//The return value is not evaluated. For a specific influence, you can also declare the

//methods explicitly and provide additional code there with the standard initialization

//code. You can evaluate the return value.
METHOD FB_Init : BOOL
VAR_INPUT
	bInitRetains : BOOL; // TRUE: the retain variables are initialized (reset warm / reset cold)
	bInCopyCode	 : BOOL; // TRUE: the instance will be copied to the copy code afterward (online change)  
	Dimensions	 : I_SingleDimensionZone;
END_VAR
_Dimensions := Dimensions;
END_METHOD

METHOD IsMoverInPosition : BOOL
VAR_INPUT
	Mover : I_XtsMover;
END_VAR

VAR
	startPosition : LREAL;
	endPosition	  : LREAL;
	tmp : LREAL;
END_VAR
startPosition := _Dimensions.StartPosition;
endPosition	  := _Dimensions.EndPosition;
IF Mover.Status.CurrentTrack.Length <> 0 THEN
	startPosition := startPosition - Mover.Status.CurrentTrack.Length * TRUNC(_Dimensions.StartPosition / Mover.Status.CurrentTrack.Length);
	IF startPosition < 0.0 THEN
		startPosition := startPosition + Mover.Status.CurrentTrack.Length;
	END_IF

	endPosition := endPosition - Mover.Status.CurrentTrack.Length * TRUNC(_Dimensions.EndPosition / Mover.Status.CurrentTrack.Length);
	IF endPosition < 0.0 THEN
		endPosition := endPosition + Mover.Status.CurrentTrack.Length;
	END_IF
END_IF

IF startPosition < endPosition THEN
	IsMoverInPosition := Mover.Position > startPosition AND Mover.Position < endPosition;
ELSE
	IsMoverInPosition := Mover.Position > startPosition OR Mover.Position < endPosition;
END_IF
END_METHOD

END_FUNCTION_BLOCK

// _Internal/Zone/Interfaces/I_MoverInPositionChecker
INTERFACE I_MoverInPositionChecker EXTENDS I_Base

METHOD IsMoverInPosition : BOOL
VAR_INPUT
	Mover : I_XtsMover;
END_VAR
END_METHOD

END_INTERFACE

// _Internal/Zone/MoverZoneDistanceComparer
{attribute 'no_explicit_call' := 'This FB is a CLASS and must be accessed using methods or properties'}
{attribute 'conditional_show'}
FUNCTION_BLOCK MoverZoneDistanceComparer IMPLEMENTS I_XtsMoverComparer
VAR
	_ZoneDimensions : I_SingleDimensionZone;
END_VAR

METHOD Compare : SINT
VAR_INPUT
	Mover1 : I_XtsMover;
	Mover2 : I_XtsMover;
END_VAR

VAR
	Mover1Distance : LREAL;
	Mover2Distance : LREAL;
END_VAR
Mover1Distance := MoverDistance(_ZoneDimensions.StartPosition, Mover1.Position, Mover1.Status.CurrentTrack.Length);
Mover2Distance := MoverDistance(_ZoneDimensions.StartPosition, Mover2.Position, Mover2.Status.CurrentTrack.Length);
IF Mover1Distance < Mover2Distance THEN
	Compare := -1;
ELSIF Mover1Distance > Mover2Distance THEN
	Compare := 1;
ELSE
	Compare := 0;
END_IF
END_METHOD

//FB_Init is always available implicitly and it is used primarily for initialization.
//The return value is not evaluated. For a specific influence, you can also declare the
//methods explicitly and provide additional code there with the standard initialization
//code. You can evaluate the return value.
METHOD FB_Init: BOOL
VAR_INPUT
    bInitRetains: BOOL; // TRUE: the retain variables are initialized (reset warm / reset cold)
    bInCopyCode: BOOL;  // TRUE: the instance will be copied to the copy code afterward (online change)   
	Dimensions : I_SingleDimensionZone;
END_VAR
_ZoneDimensions := Dimensions;
END_METHOD

END_FUNCTION_BLOCK

// _Internal/Zone/Interfaces/I_XtsMoverComparer
INTERFACE I_XtsMoverComparer EXTENDS I_Base

METHOD Compare : SINT
VAR_INPUT
	Mover1 : I_XtsMover;
	Mover2 : I_XtsMover;
END_VAR
END_METHOD

END_INTERFACE

// _Internal/Zone/MoverDistance
FUNCTION MoverDistance : LREAL
VAR_INPUT
	StartPosition : LREAL;
	MoverPosition : LREAL;
	TrackLength	  : LREAL;
END_VAR

VAR
	NormalizedStart : LREAL;
	Distance		: LREAL;
END_VAR

IF TrackLength = 0 THEN
	MoverDistance := 0;
	RETURN;
END_IF

NormalizedStart := StartPosition - TrackLength * TRUNC(StartPosition / TrackLength);
IF normalizedStart < 0 THEN
	NormalizedStart := NormalizedStart + TrackLength;
END_IF;

Distance := MoverPosition - NormalizedStart;
IF Distance < 0 THEN
	Distance := Distance + TrackLength;
END_IF;

MoverDistance := Distance;

END_FUNCTION

// _Internal/Zone/ZoneMonitor
{attribute 'no_explicit_call' := 'This FB is a CLASS and must be accessed using methods or properties'}
{attribute 'conditional_show'}
FUNCTION_BLOCK ZoneMonitor IMPLEMENTS I_ZoneMonitor
VAR
	_DefaultCurrentMovers : XtsMoverList;
	_CurrentMovers		  : I_XtsMoverList := _DefaultCurrentMovers;
	_MoverChecker		  : I_MoverInPositionChecker;
	_MonitoredMovers	  : I_XtsMoverCollection;
	_ZoneComparer		  : I_XtsMoverComparer;
	_ZoneDimensions		  : I_SingleDimensionZone;
	_Logger				  : I_MechatronicsLogger;
	LogSource			  : TraceSourceInfo;
	LogMessage			  : TraceMessageInfo;
END_VAR

METHOD CyclicLogic
VAR
	Mover				   : I_XtsMover;
	inPosition			   : BOOL;
	inCollection		   : BOOL;
	additionIndex		   : UDINT;
	CompareResults		   : SINT;
	EntranceEvent		   : E_ThresholdEvent;
	ExitEvent			   : E_ThresholdEvent;
	ThresholdEventOccurred : BOOL;
END_VAR
_MonitoredMovers.ResetIterator();
WHILE _MonitoredMovers.MoveToNext DO
	__QUERYINTERFACE(_MonitoredMovers.Current, Mover);
	IF Mover.Status.CurrentTrack.Length = 0 THEN
		LogMessage.MessageId := E_XtsLogMessage.ZoneMoverErrorTrackLengthZero;
		LogMessage.Severity	 := 3;
		_Logger.LogMessageInstance(LogSource, LogMessage);
		CONTINUE;
	END_IF

	inPosition := _MoverChecker.IsMoverInPosition(Mover);

	//Need to check if crossed the threshold of the exit or the entrance
	EntranceEvent		   := CheckForThresholdEvent(Mover, _ZoneDimensions.StartPosition);
	ExitEvent			   := CheckForThresholdEvent(Mover, _ZoneDimensions.EndPosition);
	ThresholdEventOccurred := (EntranceEvent <> E_ThresholdEvent.NoEvent) AND (ExitEvent <> E_ThresholdEvent.NoEvent);
	inCollection		   := _CurrentMovers.Contains(Mover);
	IF NOT inPosition AND inCollection THEN
		_CurrentMovers.Remove(Mover);
		CONTINUE;
	END_IF

	//Adds the Mover into the collection sorted by Position Descending
	IF inPosition AND NOT inCollection THEN
		_CurrentMovers.ResetIterator();
		WHILE _CurrentMovers.MoveToNext DO
			CompareResults := _ZoneComparer.Compare(Mover, _CurrentMovers.Current);
			IF CompareResults < 0 THEN //Mover 1 is closer to Start
				additionIndex := _CurrentMovers.CurrentItem - 1;
				EXIT;
			ELSIF CompareResults > 0 THEN //Mover 2 is closer to Start
				additionIndex := _CurrentMovers.CurrentItem;
			ELSE //Movers are equadistant, should never happen. Only realistically happens if TrackLength = 0

				//
			END_IF
		END_WHILE

		_CurrentMovers.InsertAtIndex(Mover, additionIndex);
	ELSIF ThresholdEventOccurred AND inCollection THEN
		(*Search the Collection to find the new index
			Remove from old index
			Add to new*)
		_CurrentMovers.ResetIterator();
		WHILE _CurrentMovers.MoveToNext DO
			CompareResults := _ZoneComparer.Compare(Mover, _CurrentMovers.Current);
			IF CompareResults < 0 THEN //Mover 1 is closer to Start
				additionIndex := _CurrentMovers.CurrentItem - 1;
				EXIT;
			ELSIF CompareResults > 0 THEN //Mover 2 is closer to Start
				additionIndex := _CurrentMovers.CurrentItem;
			ELSE //Movers are equadistant, should never happen. Only realistically happens if TrackLength = 0

				//
			END_IF
		END_WHILE

		_CurrentMovers.Remove(Mover);
		_CurrentMovers.InsertAtIndex(Mover, additionIndex);
	END_IF
END_WHILE
END_METHOD

//FB_Init is always available implicitly and it is used primarily for initialization.

//The return value is not evaluated. For a specific influence, you can also declare the

//methods explicitly and provide additional code there with the standard initialization

//code. You can evaluate the return value.
METHOD FB_Init : BOOL
VAR_INPUT
	bInitRetains	: BOOL; // TRUE: the retain variables are initialized (reset warm / reset cold)
	bInCopyCode		: BOOL; // TRUE: the instance will be copied to the copy code afterward (online change)   
	PositionChecker : I_MoverInPositionChecker;
	ZoneComparer	: I_XtsMoverComparer;
	ZoneDimensions	: I_SingleDimensionZone;
	Logger			: I_MechatronicsLogger;
END_VAR
_MoverChecker		 := PositionChecker;
_ZoneComparer		 := ZoneComparer;
_Logger				 := Logger;
_ZoneDimensions		 := ZoneDimensions;
LogSource.SourceName := 'ZoneMonitor';
END_METHOD

PROPERTY MonitoredMovers : I_XtsMoverCollection
SET
_MonitoredMovers := MonitoredMovers;
END_SET
END_PROPERTY

{attribute 'monitoring':='call'}
PROPERTY Movers : I_XtsMoverList
GET
Movers := _CurrentMovers;
END_GET
END_PROPERTY

END_FUNCTION_BLOCK

// _Internal/Zone/Interfaces/I_ZoneMonitor
INTERFACE I_ZoneMonitor EXTENDS I_Base, I_Cyclic, I_MonitorsMovers, I_ContainXtsMoverList

END_INTERFACE

// _Internal/Peeker/Interfaces/I_XtsModuleCollectionPeeker
INTERFACE I_XtsModuleCollectionPeeker EXTENDS I_Base

METHOD SetCollection
VAR_INPUT
	NewCollection  : I_XtsModuleCollection;
	CollectionName : T_MaxString := 'A Collection';
END_VAR
END_METHOD

END_INTERFACE

// _Internal/Peeker/Interfaces/I_XtsMoverCollectionPeeker
INTERFACE I_XtsMoverCollectionPeeker EXTENDS I_Base

METHOD SetCollection
VAR_INPUT
	NewCollection  : I_XtsMoverCollection;
	CollectionName : T_MaxString := 'A Collection';
END_VAR
END_METHOD

END_INTERFACE

// _Internal/Peeker/Interfaces/I_XtsPartCollectionPeeker
INTERFACE I_XtsPartCollectionPeeker EXTENDS I_Base

METHOD SetCollection
VAR_INPUT
	NewCollection  : I_XtsPartCollection;
	CollectionName : T_MaxString := 'A Collection';
END_VAR
END_METHOD

END_INTERFACE

// _Internal/Peeker/Interfaces/I_XtsPositionTriggerCollectionPeeker
INTERFACE I_XtsPositionTriggerCollectionPeeker EXTENDS I_Base

METHOD SetCollection
VAR_INPUT
	NewCollection  : I_XtsPositionTriggerCollection;
	CollectionName : T_MaxString := 'A Collection';
END_VAR
END_METHOD

END_INTERFACE

// _Internal/Peeker/Interfaces/I_XtsStationCollectionPeeker
INTERFACE I_XtsStationCollectionPeeker EXTENDS I_Base

METHOD SetCollection
VAR_INPUT
	NewCollection  : I_XtsStationCollection;
	CollectionName : T_MaxString := 'A Collection';
END_VAR
END_METHOD

END_INTERFACE

// _Internal/Peeker/Interfaces/I_XtsZoneCollectionPeeker
INTERFACE I_XtsZoneCollectionPeeker EXTENDS I_Base

METHOD SetCollection
VAR_INPUT
	NewCollection  : I_XtsZoneCollection;
	CollectionName : T_MaxString := 'A Collection';
END_VAR
END_METHOD

END_INTERFACE

// _Internal/Station/Interfaces/I_StationTaskCollection
INTERFACE I_StationTaskCollection EXTENDS I_Base

END_INTERFACE

// _Internal/Station/MoverMonitorTask
{attribute 'no_explicit_call' := 'This FB is a CLASS and must be accessed using methods or properties'}
FUNCTION_BLOCK MoverMonitorTask IMPLEMENTS I_MoverMonitor
VAR
	_MonitoredMovers  : I_XtsMoverCollection;
	_CurrentMover	  : I_XtsMover := NullObjects.XtsMover;
	_RemoveCollection : XtsMoverCollection;
	_Station		  : I_XtsStation;
	{attribute 'hide'}
	_Logger : I_MechatronicsLogger;
	{attribute 'hide'}
	LogSource : TraceSourceInfo;
	{attribute 'hide'}
	LogMessage : TraceMessageInfo;
END_VAR

METHOD CyclicLogic
VAR
	Mover	  : I_XtsMover;
	NullMover : I_XtsMover;
END_VAR
_MonitoredMovers.ResetIterator();
WHILE _MonitoredMovers.MoveToNext DO
	Mover := _MonitoredMovers.Current;
	IF Mover.CurrentTask.TaskId <> MoverTaskID.MOVE_TO_STATION OR Mover.Status.CommandedStation <> _Station THEN
		_RemoveCollection.AddItem(Mover);
		CONTINUE;
	END_IF

	NullMover := NullObjects.XtsMover;
	IF Mover.InPosition AND _CurrentMover = NullMover THEN
		_CurrentMover		 := Mover;
		LogMessage.Message	 := CONCAT(Mover.Name, ' arrived at station');
		LogMessage.MessageId := E_XtsLogMessage.StationMoverArrived;
		LogMessage.Severity	 := 0;
		_Logger.LogMessageInstance(LogSource, LogMessage);
		EXIT;
	END_IF
END_WHILE

IF _RemoveCollection.IsEmpty THEN
	RETURN;
END_IF

_RemoveCollection.ResetIterator();
WHILE _RemoveCollection.MoveToNext DO
	LogMessage.Message	 := CONCAT(_RemoveCollection.Current.Name, ' deregistered from Station');
	LogMessage.MessageId := E_XtsLogMessage.StationMoverDeregistered;
	LogMessage.Severity	 := 0;
	_Logger.LogMessageInstance(LogSource, LogMessage);
	IF _CurrentMover = _RemoveCollection.Current THEN
		_CurrentMover := NullObjects.XtsMover;
	END_IF

	_MonitoredMovers.Remove(_RemoveCollection.Current);
END_WHILE

IF NOT _RemoveCollection.IsEmpty THEN
	_RemoveCollection.Clear();
END_IF
END_METHOD

//FB_Init is always available implicitly and it is used primarily for initialization.

//The return value is not evaluated. For a specific influence, you can also declare the

//methods explicitly and provide additional code there with the standard initialization

//code. You can evaluate the return value.
METHOD FB_Init : BOOL
VAR_INPUT
	bInitRetains			 : BOOL; // TRUE: the retain variables are initialized (reset warm / reset cold)
	bInCopyCode				 : BOOL; // TRUE: the instance will be copied to the copy code afterward (online change)
	Station					 : I_XtsStation;
	MonitoredMoverCollection : I_XtsMoverCollection;
END_VAR
_Station		 := Station;
__QUERYINTERFACE(Station.TracePublisher,_Logger);
LogSource.SourceName := 'Mover Monitor';
_MonitoredMovers := MonitoredMoverCollection;
END_METHOD

METHOD GetMover : I_XtsMover
VAR
	NullMover : I_XtsMover;
END_VAR
NullMover := NullObjects.XtsMover;
IF _CurrentMover = NullMover THEN
	LogMessage.Message	 := 'GetMover called when no mover present.';
	LogMessage.Severity	 := 2;
	LogMessage.MessageId := E_XtsLogMessage.StationGetMoverCalledNoMover;
	_Logger.LogMessageInstance(LogSource, LogMessage);
	GetMover := NullObjects.XtsMover;
	RETURN;
END_IF

GetMover := _CurrentMover;
_MonitoredMovers.Remove(_CurrentMover);
_CurrentMover := NullObjects.XtsMover;
END_METHOD

PROPERTY MonitoredMovers : I_XtsMoverCollection
GET
MonitoredMovers := _MonitoredMovers;
END_GET
SET
_MonitoredMovers := MonitoredMovers;
END_SET
END_PROPERTY

{attribute 'monitoring':='call'}
PROPERTY MoverPresent : BOOL
GET
VAR
	NullMover : I_XtsMover;
END_VAR
NullMover	 := NullObjects.XtsMover;
MoverPresent := _CurrentMover <> NullMover;
END_GET
END_PROPERTY

END_FUNCTION_BLOCK

// _Internal/Tracing/XtsCoreEventLogger
{attribute 'no_explicit_call' := 'This FB is a CLASS and must be accessed using methods or properties'}
{attribute 'conditional_show'}
FUNCTION_BLOCK XtsCoreEventLogger IMPLEMENTS I_MechatronicsLogger
VAR
	MessagesThisScan : DINT;
	Message			 : FB_TcMessage;
	Source			 : FB_TcSourceInfo;
	CurrentCycle	 : UDINT;
END_VAR

METHOD LogMessage
VAR_INPUT
	Key		  : T_MaxString;
	Value	  : T_MaxString;
	SourceId  : UDINT := 0;
	TimeStamp : ULINT := 0;
	MessageId : UDINT := 1;
	Severity  : USINT := 1;
END_VAR

VAR_INST
	LogSource  : TraceSourceInfo;
	LogMessage : TraceMessageInfo;
END_VAR
LogSource.SourceName := Key;
LogSource.SourceId	 := SourceId;
LogSource.TimeStamp	 := TimeStamp;
LogMessage.Message	 := Value;
LogMessage.MessageId := MessageId;
LogMessage.Severity	 := Severity;
THIS^.LogMessageInstance(LogSource, LogMessage);
END_METHOD

METHOD LogMessageInstance
VAR_INPUT
	SourceInfo	: I_TraceSourceInfo;
	MessageInfo : I_TraceMessageInfo;
	Arguments	: I_TraceArgument := 0;
END_VAR
VAR
	Msg : T_MaxString;
END_VAR
IF TwinCAT_SystemInfoVarList._TaskInfo[GETCURTASKINDEXEX()].CycleCount <> CurrentCycle THEN
	CurrentCycle	 := TwinCAT_SystemInfoVarList._TaskInfo[GETCURTASKINDEXEX()].CycleCount;
	MessagesThisScan := 0;
END_IF

IF MessagesThisScan < TO_DINT(TwinCAT_SystemInfoVarList._TaskInfo[GETCURTASKINDEXEX()].CycleTime / 2000) THEN
	Source.sName := SourceInfo.SourceName;
	Source.nId	 := SourceInfo.SourceId;
	Message.Create(eventClass	:= TC_EVENT_CLASSES.XtsCoreEvents,
				   nEventId		:= MessageInfo.MessageId,
				   eSeverity	:= USINT_To_TcEventSeverity(MessageInfo.Severity),
				   ipSourceInfo := Source);

	Msg := MessageInfo.Message;
	Message.ipArguments.Clear().AddString(Msg);
	Message.Send(0);
	Message.Release();
	Source.Clear();
	MessagesThisScan := MessagesThisScan + 1;
END_IF
END_METHOD

END_FUNCTION_BLOCK

// _Internal/Zone/Properties/_DefaultZoneProperties
{attribute 'no_explicit_call' := 'This FB is a CLASS and must be accessed using methods or properties'}
FUNCTION_BLOCK _DefaultZoneProperties
VAR
	_DefaultSingleDimensionZone : SingleDimensionZone;
END_VAR

END_FUNCTION_BLOCK

// HMI/XtsModule_HMI
FUNCTION_BLOCK XtsModule_HMI EXTENDS HmiFunction
VAR
	_Module : I_XtsModule;
	{ attribute 'TcHmiSymbol.AddSymbol' }
	{ attribute 'TcHmiSymbol.AddSymbol.UserGroups' := '__SystemAdministrators,Admin' }
	Module_HMI : ST_XtsModule_HMI;
END_VAR

PROPERTY ControlObject : I_Base
SET
__QUERYINTERFACE(ControlObject, _Module);
END_SET
END_PROPERTY

METHOD CyclicLogic
IF _Module = 0 THEN
	RETURN;
END_IF

Module_HMI.ModuleReady := _Module.ModuleReady;
Module_HMI.Vdc24Okay   := _Module.Vdc24Okay;
Module_HMI.Vdc48Okay   := _Module.Vdc48Okay;
Module_HMI.Vdc24	   := _Module.Module24Vdc;
Module_HMI.Vdc48	   := _Module.Module48Vdc;
END_METHOD

(*FB_Init is always available implicitly and it is used primarily for initialization.
The return value is not evaluated. For a specific influence, you can also declare the
methods explicitly and provide additional code there with the standard initialization
code. You can evaluate the return value.*)
METHOD FB_Init : BOOL
VAR_INPUT
	(* TRUE: the retain variables are initialized (reset warm / reset cold)*)
	bInitRetains : BOOL;

	(* TRUE: the instance will be copied to the copy code afterward (online change)   *)
	bInCopyCode : BOOL;
	Name		: Core.T_MaxString;
	XtsModule	: I_XtsModule;
END_VAR
THIS^._Module	:= XtsModule;
ControlType		:= 'XtsModule';
LinkObject		:= 'Module_HMI';
Module_HMI.Name := XtsModule.Name;
END_METHOD

PROPERTY XtsModule : I_XtsModule
SET
_Module			:= XtsModule;
Module_Hmi.Name := _Module.Name;
END_SET
END_PROPERTY

END_FUNCTION_BLOCK

// HMI/XtsMover_HMI
FUNCTION_BLOCK XtsMover_HMI EXTENDS HmiFunction
VAR
	Mover : I_XtsMover;
	{ attribute 'TcHmiSymbol.AddSymbol' }
	{ attribute 'TcHmiSymbol.AddSymbol.UserGroups' := '__SystemAdministrators,Admin' }
	Mover_HMI : ST_XtsMover_HMI;
END_VAR

PROPERTY ControlObject : I_Base
SET
__QUERYINTERFACE(ControlObject, Mover);
END_SET
END_PROPERTY

METHOD CyclicLogic
VAR_INST
	ClearLogRT		 : R_TRIG;
END_VAR
IF Mover = 0 THEN
	RETURN;
END_IF

Mover_HMI.Position		:= Mover.Position;
Mover_HMI.Id			:= Mover.MoverId;
Mover_HMI.LocalLog.Logs := Mover.CommandLog.Commands;
ClearLogRT(Clk := Mover_HMI.LocalLog.ClearLog);
IF ClearLogRT.Q THEN
	Mover.CommandLog.Clear();
END_IF
END_METHOD

(*FB_Init is always available implicitly and it is used primarily for initialization.
The return value is not evaluated. For a specific influence, you can also declare the
methods explicitly and provide additional code there with the standard initialization
code. You can evaluate the return value.*)
METHOD FB_Init : BOOL
VAR_INPUT
	(* TRUE: the retain variables are initialized (reset warm / reset cold)*)
	bInitRetains : BOOL;

	(* TRUE: the instance will be copied to the copy code afterward (online change)   *)
	bInCopyCode : BOOL;
	Name		: Core.T_MaxString;
	Mover		: I_XtsMover;
END_VAR
THIS^.Mover	  := Mover;
ControlType	  := 'XtsMover';
LinkObject	  := 'Mover_HMI';
Mover_HMI.Name := Mover.Name;
END_METHOD

PROPERTY XtsMover : I_XtsMover
SET
Mover := XtsMover;
Mover_Hmi.Name := Mover.Name;
END_SET
END_PROPERTY

END_FUNCTION_BLOCK

// HMI/XtsPart_HMI
FUNCTION_BLOCK XtsPart_HMI EXTENDS HmiFunction
VAR
	Part : I_XtsPart;
	{ attribute 'TcHmiSymbol.AddSymbol' }
	{ attribute 'TcHmiSymbol.AddSymbol.UserGroups' := '__SystemAdministrators,Admin' }
	Part_HMI : ST_XtsPart_HMI;
END_VAR

PROPERTY ControlObject : I_Base
SET
__QUERYINTERFACE(ControlObject, Part);
END_SET
END_PROPERTY

METHOD CyclicLogic
IF Part = 0 THEN
	RETURN;
END_IF

Part_HMI.NumberOfModules := Part.NumberModulesNotReady + Part.NumberModulesReady;
Part_HMI.PartReady		 := Part.PartReady;
Part_HMI.Id				 := Part.XtsPartId;
Part_HMI.Vdc24Okay		 := Part.Vdc24Okay;
Part_HMI.Vdc48Okay		 := Part.Vdc48Okay;
END_METHOD

(*FB_Init is always available implicitly and it is used primarily for initialization.
The return value is not evaluated. For a specific influence, you can also declare the
methods explicitly and provide additional code there with the standard initialization
code. You can evaluate the return value.*)
METHOD FB_Init : BOOL
VAR_INPUT
	(* TRUE: the retain variables are initialized (reset warm / reset cold)*)
	bInitRetains : BOOL;

	(* TRUE: the instance will be copied to the copy code afterward (online change)   *)
	bInCopyCode : BOOL;
	Name		: Core.T_MaxString;
	Part		: I_XtsPart;
END_VAR
THIS^.Part	  := Part;
ControlType	  := 'XtsPart';
LinkObject	  := 'Part_HMI';
Part_HMI.Name := Part.Name;
END_METHOD

PROPERTY XtsPart : I_XtsPart
SET
Part := XtsPart;
Part_HMI.Name := Part.Name;
END_SET
END_PROPERTY

END_FUNCTION_BLOCK

// HMI/XtsPositionTrigger_HMI
FUNCTION_BLOCK XtsPositionTrigger_HMI EXTENDS HmiFunction
VAR
	PositionTrigger : I_XtsPositionTrigger;
	{ attribute 'TcHmiSymbol.AddSymbol' }
	{ attribute 'TcHmiSymbol.AddSymbol.UserGroups' := '__SystemAdministrators,Admin' }
	PositionTrigger_HMI : ST_XtsPositionTrigger_HMI;
END_VAR

PROPERTY ControlObject : I_Base
SET
__QUERYINTERFACE(ControlObject, PositionTrigger);
END_SET
END_PROPERTY

METHOD CyclicLogic
VAR_INST
	EnableRT   : R_TRIG;
	DisableRT  : R_TRIG;
	ClearLogRT : R_TRIG;
END_VAR
IF PositionTrigger = 0 THEN
	RETURN;
END_IF

PositionTrigger_HMI.Enabled				   := PositionTrigger.Enabled;
PositionTrigger_HMI.MoverPresent		   := PositionTrigger.MoverIsPresent;
PositionTrigger_HMI.NumberMoversRegistered := PositionTrigger.Status.NumberOfMoversRegistered;
PositionTrigger_HMI.Position			   := PositionTrigger.Position;
PositionTrigger_HMI.LocalLog.Logs		   := PositionTrigger.CommandLog.Commands;
PositionTrigger_HMI.NumberEventsInQueue	   := PositionTrigger.MoverQueue.Count;
ClearLogRT(Clk := PositionTrigger_HMI.LocalLog.ClearLog);
IF ClearLogRT.Q THEN
	PositionTrigger.CommandLog.Clear();
END_IF

EnableRT(Clk := PositionTrigger_HMI.Enable);
IF NOT PositionTrigger_HMI.Enabled AND EnableRT.Q THEN
	PositionTrigger.Enable();
END_IF

DisableRT(Clk := PositionTrigger_HMI.Disable);
IF PositionTrigger_HMI.Enabled AND DisableRT.Q THEN
	PositionTrigger.Disable();
END_IF
END_METHOD

(*FB_Init is always available implicitly and it is used primarily for initialization.
The return value is not evaluated. For a specific influence, you can also declare the
methods explicitly and provide additional code there with the standard initialization
code. You can evaluate the return value.*)
METHOD FB_Init : BOOL
VAR_INPUT
	(* TRUE: the retain variables are initialized (reset warm / reset cold)*)
	bInitRetains : BOOL;

	(* TRUE: the instance will be copied to the copy code afterward (online change)   *)
	bInCopyCode		: BOOL;
	Name			: Core.T_MaxString;
	PositionTrigger : I_XtsPositionTrigger;
END_VAR
THIS^.PositionTrigger	 := PositionTrigger;
ControlType				 := 'XtsPositionTrigger';
LinkObject				 := 'PositionTrigger_HMI';
PositionTrigger_HMI.Name := PositionTrigger.Name;
END_METHOD

PROPERTY XtsPositionTrigger : I_XtsPositionTrigger
SET
PositionTrigger := XtsPositionTrigger;
PositionTrigger_HMI.Name := PositionTrigger.Name;
END_SET
END_PROPERTY

END_FUNCTION_BLOCK

// HMI/XtsStation_HMI
{attribute 'enable_dynamic_creation'}
FUNCTION_BLOCK XtsStation_HMI EXTENDS HmiFunction
VAR
	Station : I_XtsStation;
	{ attribute 'TcHmiSymbol.AddSymbol' }
	{ attribute 'TcHmiSymbol.AddSymbol.UserGroups' := '__SystemAdministrators,Admin' }
	Station_HMI : ST_XtsStation_HMI;
END_VAR

PROPERTY ControlObject : I_Base
SET
__QUERYINTERFACE(ControlObject, Station);
END_SET
END_PROPERTY

METHOD CyclicLogic
VAR_INST
	EnableRT   : R_TRIG;
	DisableRT  : R_TRIG;
	ClearLogRT : R_TRIG;
END_VAR
IF Station = 0 THEN
	RETURN;
END_IF

Station_HMI.Enabled				   := Station.Enabled;
Station_HMI.MoverPresent		   := Station.MoverIsPresent;
Station_HMI.NumberMoversRegistered := Station.Status.NumberOfMoversRegistered;
Station_HMI.Position			   := Station.Position;
Station_HMI.LocalLog.Logs		   := Station.CommandLog.Commands;
ClearLogRT(Clk := Station_HMI.LocalLog.ClearLog);
IF ClearLogRT.Q THEN
	Station.CommandLog.Clear();
END_IF

EnableRT(Clk := Station_HMI.Enable);
IF NOT Station_HMI.Enabled AND EnableRT.Q THEN
	Station.Enable();
END_IF

DisableRT(Clk := Station_HMI.Disable);
IF Station_HMI.Enabled AND DisableRT.Q THEN
	Station.Disable();
END_IF
END_METHOD

(*FB_Init is always available implicitly and it is used primarily for initialization.
The return value is not evaluated. For a specific influence, you can also declare the
methods explicitly and provide additional code there with the standard initialization
code. You can evaluate the return value.*)
METHOD FB_Init : BOOL
VAR_INPUT
	(* TRUE: the retain variables are initialized (reset warm / reset cold)*)
	bInitRetains : BOOL;

	(* TRUE: the instance will be copied to the copy code afterward (online change)   *)
	bInCopyCode : BOOL;
	Name		: Core.T_MaxString;
	Station		: I_XtsStation;
END_VAR
THIS^.Station	 := Station;
ControlType		 := 'XtsStation';
LinkObject		 := 'Station_HMI';
Station_HMI.Name := Station.Name;
END_METHOD

PROPERTY XtsStation : I_XtsStation
SET
Station := XtsStation;
Station_HMI.Name := Station.Name;
END_SET
END_PROPERTY

END_FUNCTION_BLOCK

// XtsStation/XtsStation
{attribute 'no_explicit_call' := 'This FB is a CLASS and must be accessed using methods or properties'}
FUNCTION_BLOCK XtsStation EXTENDS CyclicComponent IMPLEMENTS I_Base, I_XtsStation
VAR
	{attribute 'hide'}
	_Enabled : BOOL;
	{attribute 'hide'}
	_DefaultMoverlistBehavior : XtsMoverCollection;
	_RegisteredMovers		  : I_XtsMoverCollection := _DefaultMoverlistBehavior;
	{attribute 'hide'}
	_Status : XtsStationStatus(THIS^, _DefaultMoverMonitor);

	//
	_DefaultPositionBehavior : ReferencedPosition;
	_Position				 : I_Positionable := _DefaultPositionBehavior;

	//
	_DefaultMoverMonitor : MoverMonitorTask(THIS^, _RegisteredMovers);
	_MoverMonitor		 : I_MoverMonitor := _DefaultMoverMonitor;
	{attribute 'hide'}
	_LocalLogger : MechatronicsLocalLogger;
	{attribute 'hide'}
	_Logger : MechatronicsTracePublisher;
	{attribute 'hide'}
	LogMessage : TraceMessageInfo;
	{attribute 'hide'}
	LogSource : TraceSourceInfo;
END_VAR

//FB_Init is always available implicitly and it is used primarily for initialization.

//The return value is not evaluated. For a specific influence, you can also declare the

//methods explicitly and provide additional code there with the standard initialization

//code. You can evaluate the return value.
METHOD FB_Init : BOOL
VAR_INPUT
	bInitRetains : BOOL;				 // TRUE: the retain variables are initialized (reset warm / reset cold)
	bInCopyCode	 : BOOL;				 // TRUE: the instance will be copied to the copy code afterward (online change)
	Name		 : T_MaxString;			 //Name of the Station
	Position	 : LREAL;				 //Position in mm the Station will be located
	System		 : I_ContainXtsStations; //XtsSystem to self register to
END_VAR
_Position.Position	 := Position;
LogSource.SourceName := Name;
IF System <> 0 THEN
	System.Stations.AddItem(THIS^);
	RegisterWithParent(System);
END_IF

_Status.SetRegisteredMovers(_RegisteredMovers);
_Logger.Subscribe(_LocalLogger);
IF XtsCoreParameters.TcEventLoggerEnabled THEN
	_Logger.Subscribe(XtsTrace.EventLogger);
END_IF
END_METHOD

//Disable the station
METHOD Disable
VAR
	LogMessage : TraceMessageInfo;
	LogSource  : TraceSourceInfo;
END_VAR
_Enabled := FALSE;
LogSource.SourceName := _Name;
LogMessage.Message	 := 'Disabled.';
LogMessage.MessageId := E_XtsLogMessage.StationDisabled;
_Logger.LogMessageInstance(LogSource, LogMessage);
END_METHOD

//Enable the station
METHOD Enable
VAR
	LogMessage : TraceMessageInfo;
	LogSource  : TraceSourceInfo;
END_VAR
_Enabled			 := TRUE;
LogSource.SourceName := _Name;
LogMessage.Message	 := 'Enabled.';
LogMessage.MessageId := E_XtsLogMessage.StationEnabled;
_Logger.LogMessageInstance(LogSource, LogMessage);
END_METHOD

{attribute 'monitoring' := 'call'}
PROPERTY Enabled : BOOL
GET
Enabled := _Enabled;
END_GET
END_PROPERTY

{attribute 'monitoring':='call'}
PROPERTY CommandLog : I_MechatronicsLocalLog
GET
CommandLog := _LocalLogger;
END_GET
END_PROPERTY

PROPERTY TracePublisher : I_MechatronicsTracePublisher
GET
TracePublisher := _Logger;
END_GET
END_PROPERTY

METHOD AcceptStationVisitor
VAR_INPUT
	StationVisitor : I_XtsStationVisitor;
END_VAR
StationVisitor.VisitStation(THIS^);
END_METHOD

METHOD CyclicLogic
IF NOT _Enabled THEN
	RETURN;
END_IF
_MoverMonitor.CyclicLogic();
END_METHOD

//Deregisters Mover to be Monitored by Station
METHOD DeregisterMover
VAR_INPUT
	Mover : I_XtsMover; //Mover to Deregister
END_VAR
_RegisteredMovers.Remove(Mover);
LogSource.SourceName := _Name;
LogMessage.Message	 := CONCAT('Mover Deregistered: ', Mover.Name);
LogMessage.Severity	 := 0;
LogMessage.MessageId := E_XtsLogMessage.StationMoverDeregistered;
_Logger.LogMessageInstance(LogSource, LogMessage);
END_METHOD

//Gets the Current Mover latched at the Station
METHOD GetMover : I_XtsMover
VAR_INPUT
END_VAR

VAR
	_Mover	   : I_XtsMover;
	LogMessage : TraceMessageInfo;
	LogSource  : TraceSourceInfo;
END_VAR
_Mover				 := _MoverMonitor.GetMover();
LogSource.SourceName := _Name;
LogMessage.Message	 := CONCAT('Get Mover called: ', _Mover.Name);
LogMessage.Severity	 := 10;
LogMessage.MessageId := E_XtsLogMessage.StationGetMoverCalled;
_Logger.LogMessageInstance(LogSource, LogMessage);
GetMover := _Mover;
END_METHOD

//Checks if provided Mover is registered and monitored
METHOD IsMoverRegistered : BOOL
VAR_INPUT
	Mover : I_XtsMover; //Mover to check
END_VAR
_RegisteredMovers.ResetIterator();
WHILE _RegisteredMovers.MoveToNext DO
	IF _RegisteredMovers.Current = Mover THEN
		IsMoverRegistered := TRUE;
		RETURN;
	END_IF
END_WHILE
END_METHOD

{attribute 'monitoring' := 'call'}
//Signal for if a Mover has arrived at the Station.
PROPERTY MoverIsPresent : BOOL
GET
MoverIsPresent := _MoverMonitor.MoverPresent;
END_GET
END_PROPERTY

//Currently registered and monitored Movers
PROPERTY Movers : I_XtsMoverEnumerator
GET
Movers := _RegisteredMovers;
END_GET
END_PROPERTY

{attribute 'monitoring' := 'call'}
//Location of the Station in mm
PROPERTY Position : LREAL
GET
Position := _Position.Position;
END_GET
SET
_Position.Position := Position;
END_SET
END_PROPERTY

//Registers Mover to be Monitored by Station
METHOD RegisterMover
VAR_INPUT
	Mover : I_XtsMover; //Mover to regsiter
END_VAR

VAR
	found	   : BOOL;
END_VAR
_RegisteredMovers.ResetIterator();
WHILE _RegisteredMovers.MoveToNext DO
	found := _RegisteredMovers.Current = Mover;
	IF found THEN
		RETURN;
	END_IF
END_WHILE

_RegisteredMovers.AddItem(Mover);
LogSource.SourceName := _Name;
LogMessage.Message	 := CONCAT('Mover Registered: ', Mover.Name);
LogMessage.Severity	 := 0;
LogMessage.MessageId := E_XtsLogMessage.StationMoverRegistered;
_Logger.LogMessageInstance(LogSource, LogMessage);
END_METHOD

{attribute 'monitoring':='call'}
PROPERTY Status : I_XtsStationStatus
GET
Status := _Status;
END_GET
END_PROPERTY

END_FUNCTION_BLOCK

// HMI/XtsSystem_HMI
FUNCTION_BLOCK XtsSystem_HMI EXTENDS HmiFunction
VAR
	System : I_XtsSystem;
	{ attribute 'TcHmiSymbol.AddSymbol' }
	{ attribute 'TcHmiSymbol.AddSymbol.UserGroups' := '__SystemAdministrators,Admin' }
	System_HMI : ST_XtsSystem_HMI;
END_VAR

PROPERTY ControlObject : I_Base
SET
__QUERYINTERFACE(ControlObject, System);
END_SET
END_PROPERTY

METHOD CyclicLogic
VAR_INST
	ClearLogRT		 : R_TRIG;
END_VAR
IF System = 0 THEN
	RETURN;
END_IF

System_HMI.MoverType				:= System.UtilityProperties.Mover.XtsMoverType;
System_HMI.NumberOfStations			:= System.Status.NumberOfStations;
System_HMI.NumberOfPositionTriggers := System.Status.NumberOfPositionTriggers;
System_HMI.NumberOfMovers			:= System.Status.NumberOfMovers;
System_HMI.NumberOfParts			:= System.Status.NumberOfParts;
System_HMI.NumberOfTracks			:= System.Status.NumberOfTracks;
System_HMI.NumberOfZones			:= System.Status.NumberOfZones;
System_HMI.Simulated				:= System.Status.Simulated;
System_HMI.Vdc24Okay				:= System.Status.Vdc24Okay;
System_HMI.Vdc48Okay				:= System.Status.Vdc48Okay;
System_HMI.LocalLog.Logs			:= System.CommandLog.Commands;
ClearLogRT(Clk := System_HMI.LocalLog.ClearLog);
IF ClearLogRT.Q THEN
	System.CommandLog.Clear();
END_IF
END_METHOD

(*FB_Init is always available implicitly and it is used primarily for initialization.
The return value is not evaluated. For a specific influence, you can also declare the
methods explicitly and provide additional code there with the standard initialization
code. You can evaluate the return value.*)
METHOD FB_Init : BOOL
VAR_INPUT
	(* TRUE: the retain variables are initialized (reset warm / reset cold)*)
	bInitRetains : BOOL;

	(* TRUE: the instance will be copied to the copy code afterward (online change)   *)
	bInCopyCode : BOOL;
	Name		: Core.T_MaxString;
	System		: I_XtsSystem;
END_VAR
THIS^.System	  := System;
ControlType	  := 'XtsSystem';
LinkObject	  := 'System_HMI';
System_HMI.Name := System.Name;
END_METHOD

END_FUNCTION_BLOCK

// HMI/XtsZone_HMI
FUNCTION_BLOCK XtsZone_HMI EXTENDS HmiFunction
VAR
	Zone : I_XtsZone;
	{ attribute 'TcHmiSymbol.AddSymbol' }
	{ attribute 'TcHmiSymbol.AddSymbol.UserGroups' := '__SystemAdministrators,Admin' }
	Zone_HMI : ST_XtsZone_HMI;
END_VAR

PROPERTY ControlObject : I_Base
SET
__QUERYINTERFACE(ControlObject, Zone);
END_SET
END_PROPERTY

METHOD CyclicLogic
VAR_INST
	SortedMoverRT	 : R_TRIG;
	ClearLogRT		 : R_TRIG;
END_VAR
IF Zone = 0 THEN
	RETURN;
END_IF

Zone_HMI.StartPosition		:= Zone.StartPosition;
Zone_HMI.EndPosition		:= Zone.EndPosition;
Zone_HMI.NumberMoversInZone := Zone.Status.NumberOfMoversInZone;
ClearLogRT(Clk := Zone_HMI.LocalLog.ClearLog);
IF ClearLogRT.Q THEN
	Zone.CommandLog.Clear();
END_IF

SortedMoverRT(Clk := Zone_HMI.GetSortedMover);
IF SortedMoverRT.Q THEN
	Zone_HMI.SortedMover := Zone.GetSortedMover(Zone_Hmi.SortedPosition, Zone_Hmi.SortedDirection).Name;
END_IF
END_METHOD

(*FB_Init is always available implicitly and it is used primarily for initialization.
The return value is not evaluated. For a specific influence, you can also declare the
methods explicitly and provide additional code there with the standard initialization
code. You can evaluate the return value.*)
METHOD FB_Init : BOOL
VAR_INPUT
	(* TRUE: the retain variables are initialized (reset warm / reset cold)*)
	bInitRetains : BOOL;

	(* TRUE: the instance will be copied to the copy code afterward (online change)   *)
	bInCopyCode : BOOL;
	Name		: Core.T_MaxString;
	Zone		: I_XtsZone;
END_VAR
THIS^.Zone	  := Zone;
ControlType	  := 'XtsZone';
LinkObject	  := 'Zone_HMI';
Zone_HMI.Name := Zone.Name;
END_METHOD

END_FUNCTION_BLOCK

// Project Information/F_GetCompany
// This function has been automatically generated from the project information.
{attribute 'signature_flag' := '1073741824'}
{attribute 'TcGenerated'}
{attribute 'no-analysis'}
FUNCTION F_GetCompany : WSTRING
VAR_INPUT
	
END_VAR

F_GetCompany := "Beckhoff Automation LLC";

END_FUNCTION

// Project Information/F_GetTitle
// This function has been automatically generated from the project information.
{attribute 'signature_flag' := '1073741824'}
{attribute 'TcGenerated'}
{attribute 'no-analysis'}
FUNCTION F_GetTitle : WSTRING
VAR_INPUT
	
END_VAR

F_GetTitle := "XtsCore";

END_FUNCTION

// Project Information/F_GetVersion
// This function has been automatically generated from the project information.
{attribute 'signature_flag' := '1073741824'}
{attribute 'TcGenerated'}
{attribute 'no-analysis'}
FUNCTION F_GetVersion : ST_LibVersion
VAR_INPUT
	
END_VAR

F_GetVersion.iMajor := 0;
F_GetVersion.iMinor := 9;
F_GetVersion.iBuild := 5;
F_GetVersion.iRevision := 1;
F_GetVersion.sVersion := '0.9.5.1';
F_GetVersion.nFlags := 0;

END_FUNCTION

// Utilities/IsNullObject
FUNCTION IsNullObject : BOOL
VAR_INPUT
	Object : I_Base;
END_VAR
VAR
	NullObject : I_NullObject;
END_VAR

IsNullObject := __QUERYINTERFACE(Object,NullObject);

END_FUNCTION

// Utilities/IsValidObject
FUNCTION IsValidObject : BOOL
VAR_INPUT
	Object : I_Base;
END_VAR
VAR
	value : BOOL;
	inverse : BOOL;
	NullObject : I_NullObject;
END_VAR

IsValidObject := (NOT __QUERYINTERFACE(Object, NullObject));

END_FUNCTION

// XtsStation/Interfaces/I_MoverPositionMonitor
INTERFACE I_MoverPositionMonitor EXTENDS I_Base

END_INTERFACE
